INTERFACE I_ComponentsCollection

METHOD PUBLIC AddComponent : BOOL
VAR_INPUT
    newComponent : I_ComponentBase;
END_VAR
END_METHOD

METHOD PUBLIC ContainsComponent : BOOL
VAR_INPUT
    newComponent : I_ComponentBase;
END_VAR
END_METHOD

PROPERTY Count : UINT
GET
END_GET
END_PROPERTY

METHOD PUBLIC CyclicLogic
VAR_INPUT
END_VAR
END_METHOD

METHOD PUBLIC GetComponent : BOOL
VAR_INPUT
    index : UDINT;
END_VAR
END_METHOD

METHOD PUBLIC Initialize
VAR_INPUT
END_VAR
END_METHOD

METHOD PUBLIC RemoveComponent : BOOL
VAR_INPUT
    newComponent : I_ComponentBase;
END_VAR
END_METHOD

METHOD PUBLIC RemoveComponentAt : BOOL
VAR_INPUT
    index : UDINT;
END_VAR
END_METHOD

END_INTERFACE

(* stored: Version 1.1.0.1, ProductVersion 3.1.4024.12
   Itf I_ComponentsCollection: Id {cd9c2909-80e7-4016-b04d-a23c195a6ce8}
   Method AddComponent: Id {83e1e1b6-7c85-4e2a-abd1-4d9b2ad23b80}
   Method ContainsComponent: Id {a0cf17a4-8017-483f-9a01-73fbb07c1228}
   Property Count: Id {fe986b55-8778-4207-bff0-0f1653e15d28}
   Get Get: Id {4ed50cef-02d5-42d1-b4fd-b0619b4c958b}
   Method CyclicLogic: Id {9a5a3925-2d2b-42a3-a404-328faeabd89d}
   Method GetComponent: Id {ba6631e6-fe35-42d5-b7b5-60e13f7db048}
   Method Initialize: Id {aeb5ced7-24f3-46b2-b410-ed376d31c453}
   Method RemoveComponent: Id {4f7f742f-42b2-49be-8427-666df7448bab}
   Method RemoveComponentAt: Id {4ed8bee8-b38f-44ef-be81-4672323043ad} *)
